// TIA Portal V20 export
DATA_BLOCK "OPC_Data"   // DB41
// stored: MemoryReserve 0, Namespace ProductionLine
   VAR
      Watchdog : Struct
         Keep_Alive_PLC : Int;   // //Periodic counter, incremented every 10 seconds. If one side does not increment the counter within 30 seconds, it will be considered offline by the other side.
         Keep_Alive_WMS : Int;   // //Periodic counter, incremented every 10 seconds. If one side does not increment the counter within 30 seconds, it will be considered offline by the other side.
      END_STRUCT;
      DP1 : Struct
         DestRequest : Struct
            Source : "ProductionLine.OPC_DsetRequest";
            Ack { S7_SetPoint := 'True'} : "ProductionLine.OPC_DestRequest_Ack";
         END_STRUCT;
      END_STRUCT;
      DP2 : Struct
         DestRequest : Struct
            Source : "ProductionLine.OPC_DsetRequest";
            Ack { S7_SetPoint := 'True'} : "ProductionLine.OPC_DestRequest_Ack";
         END_STRUCT;
      END_STRUCT;
      DP3 : Struct
         DestRequest : Struct
            Source : "ProductionLine.OPC_DsetRequest";
            Ack { S7_SetPoint := 'True'} : "ProductionLine.OPC_DestRequest_Ack";
         END_STRUCT;
      END_STRUCT;
      DP4 : Struct
         DestRequest : Struct
            Source : "ProductionLine.OPC_DsetRequest";
            Ack { S7_SetPoint := 'True'} : "ProductionLine.OPC_DestRequest_Ack";
         END_STRUCT;
      END_STRUCT;
      IP11 : Struct
         DestInfo : Struct
            Source : "ProductionLine.OPC_DestInfo";
            Ack { S7_SetPoint := 'True'} : "ProductionLine.OPC_DestInfo_Ack";
         END_STRUCT;
      END_STRUCT;
      IP12 : Struct
         DestInfo : Struct
            Source : "ProductionLine.OPC_DestInfo";
            Ack { S7_SetPoint := 'True'} : "ProductionLine.OPC_DestInfo_Ack";
         END_STRUCT;
      END_STRUCT;
      IP21 : Struct
         DestInfo : Struct
            Source : "ProductionLine.OPC_DestInfo";
            Ack { S7_SetPoint := 'True'} : "ProductionLine.OPC_DestInfo_Ack";
         END_STRUCT;
      END_STRUCT;
      IP22 : Struct
         DestInfo : Struct
            Source : "ProductionLine.OPC_DestInfo";
            Ack { S7_SetPoint := 'True'} : "ProductionLine.OPC_DestInfo_Ack";
         END_STRUCT;
      END_STRUCT;
      IP23 : Struct
         DestInfo : Struct
            Source : "ProductionLine.OPC_DestInfo";
            Ack { S7_SetPoint := 'True'} : "ProductionLine.OPC_DestInfo_Ack";
         END_STRUCT;
      END_STRUCT;
      IP31 : Struct
         DestInfo : Struct
            Source : "ProductionLine.OPC_DestInfo";
            Ack { S7_SetPoint := 'True'} : "ProductionLine.OPC_DestInfo_Ack";
         END_STRUCT;
      END_STRUCT;
      IP32 : Struct
         DestInfo : Struct
            Source : "ProductionLine.OPC_DestInfo";
            Ack { S7_SetPoint := 'True'} : "ProductionLine.OPC_DestInfo_Ack";
         END_STRUCT;
      END_STRUCT;
      IP41 : Struct
         DestInfo : Struct
            Source : "ProductionLine.OPC_DestInfo";
            Ack { S7_SetPoint := 'True'} : "ProductionLine.OPC_DestInfo_Ack";
         END_STRUCT;
      END_STRUCT;
      IP42 : Struct
         DestInfo : Struct
            Source : "ProductionLine.OPC_DestInfo";
            Ack { S7_SetPoint := 'True'} : "ProductionLine.OPC_DestInfo_Ack";
         END_STRUCT;
      END_STRUCT;
      Status : "ProductionLine.OPC_SegmentStatus";
   END_VAR
BEGIN
   DP1.DestRequest.Source.DecisionPoint := 'DP1';
   DP2.DestRequest.Source.DecisionPoint := 'DP2';
   DP3.DestRequest.Source.DecisionPoint := 'DP3';
   DP4.DestRequest.Source.DecisionPoint := 'DP4';
   IP11.DestInfo.Source.DecisionPoint := 'DP1';
   IP12.DestInfo.Source.DecisionPoint := 'DP1';
   IP21.DestInfo.Source.DecisionPoint := 'DP2';
   IP22.DestInfo.Source.DecisionPoint := 'DP2';
   IP23.DestInfo.Source.DecisionPoint := 'DP2';
   IP31.DestInfo.Source.DecisionPoint := 'DP3';
   IP32.DestInfo.Source.DecisionPoint := 'DP3';
   IP41.DestInfo.Source.DecisionPoint := 'DP4';
   IP42.DestInfo.Source.DecisionPoint := 'DP4';
END_DATA_BLOCK
